ADAPTER WagoRegCom (* Register communication for Wago modules *)
  (* Standard: 61499-2; Description: Copyright (c) 2026 Monika Wenger This program and the accompanying materials are made available under the terms of the Eclipse Public License 2.0 which is available at https://www.eclipse.org/legal/epl-2.0/ SPDX-License-Identifier: EPL-2.0 *)
  (* Version 3.0, 2026-07-21, Monika Wenger *)
  PACKAGE eclipse4diac::io::wago;
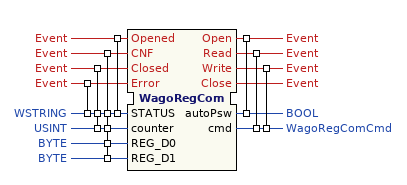
  EVENT_INPUT
    Opened WITH STATUS; (* Confirms opening of register communication *)
    CNF WITH counter, REG_D0, REG_D1, STATUS; (* Confirms that the R/W command has been processed *)
    Closed WITH STATUS, counter; (* Confirms closing of register communication *)
    Error WITH STATUS; (* Indicates errors *)
  END_EVENT
  EVENT_OUTPUT
    Open WITH autoPsw; (* Open register communication *)
    Read WITH cmd; (* Read register with RegNr *)
    Write WITH cmd; (* Write register with RegNr *)
    Close; (* Close register communication *)
  END_EVENT
  VAR_INPUT
    STATUS : WSTRING; (* Status message *)
    counter : USINT; (* Counts the commands processed *)
    REG_D0 : BYTE; (* LSB data read from the register RegNr of the cmd *)
    REG_D1 : BYTE; (* MSB data read from the register RegNr of the cmd *)
  END_VAR
  VAR_OUTPUT
    autoPsw : BOOL := TRUE; (* Automatically (re)sets password to write secured registers *)
    cmd : eclipse4diac::io::wago::WagoRegComCmd; (* Command for register communication *)
  END_VAR
END_ADAPTER
